TYPE
    ST_Auto_Storage :
    STRUCT
    END_STRUCT
END_TYPE

(* stored: Version 1.1.0.1, ProductVersion 3.1.4024.13
   DUT ST_Auto_Storage: Id {3ad64069-c854-418d-907a-eae86045a419} *)
